INTERFACE I_PressureGroup

PROPERTY bPressureHigh : BOOL
GET
END_GET
END_PROPERTY

PROPERTY bPressureLow : BOOL
GET
END_GET
END_PROPERTY

PROPERTY fScaledPressureValue : REAL
GET
END_GET
END_PROPERTY

END_INTERFACE

(* stored: Version 1.1.0.1
   Itf I_PressureGroup: Id {1e361af1-eb81-0639-2540-caa4315fac07}
   Property bPressureHigh: Id {71df05fc-5032-0c63-3f95-2e923ef5c275}
   Get Get: Id {f0ba445a-7413-0135-0268-37b377e91c05}
   Property bPressureLow: Id {f249617a-6bcf-02dc-10de-eb7be8179edb}
   Get Get: Id {81528a58-bd64-05e1-32cd-7952bd8bf52a}
   Property fScaledPressureValue: Id {ddf1f188-a4db-0c49-1996-48d24cb2467c}
   Get Get: Id {cf025ad1-5fda-0c97-2075-07e2f62da985} *)
